(* IEC 61131-3 sources: STruCpp/tests/st-validation/function_blocks, 40 files *)

(* ---- basic_fb.st ---- *)
FUNCTION_BLOCK Counter
  VAR_INPUT increment : INT; END_VAR
  VAR_OUTPUT count : INT; END_VAR
  count := count + increment;
END_FUNCTION_BLOCK

FUNCTION_BLOCK Toggle
  VAR_OUTPUT state : BOOL; END_VAR
  state := NOT state;
END_FUNCTION_BLOCK

(* ---- fb_abstract.st ---- *)
FUNCTION_BLOCK ABSTRACT Shape
  VAR_OUTPUT area : REAL; END_VAR

  METHOD PUBLIC ABSTRACT GetArea : REAL
  END_METHOD
END_FUNCTION_BLOCK

FUNCTION_BLOCK Circle EXTENDS Shape
  VAR_INPUT radius : REAL; END_VAR

  METHOD PUBLIC GetArea : REAL
    GetArea := 3.14159 * radius * radius;
  END_METHOD

  area := THIS.GetArea();
END_FUNCTION_BLOCK

(* ---- fb_accumulator.st ---- *)
FUNCTION_BLOCK AccumulatorFB
  VAR_INPUT inc : INT; END_VAR
  VAR total : INT; END_VAR
  VAR_OUTPUT result : INT; END_VAR
  total := total + inc;
  result := total;
END_FUNCTION_BLOCK

(* ---- fb_composition.st ---- *)
FUNCTION_BLOCK Sensor
  VAR_OUTPUT value : INT; END_VAR
  value := 42;
END_FUNCTION_BLOCK

FUNCTION_BLOCK Controller
  VAR
    sensor : Sensor;
    reading : INT;
    processed : BOOL;
  END_VAR
  sensor();
  reading := sensor.value;
  processed := TRUE;
END_FUNCTION_BLOCK

(* ---- fb_constructor_defaults.st ---- *)
FUNCTION_BLOCK ConfigFB
  VAR_INPUT
    maxCount : INT;
  END_VAR
  VAR_OUTPUT
    ready : BOOL;
  END_VAR
  VAR
    counter : INT;
  END_VAR
  IF counter < maxCount THEN
    counter := counter + 1;
  END_IF;
  ready := counter >= maxCount;
END_FUNCTION_BLOCK

(* ---- fb_deep_method.st ---- *)
FUNCTION_BLOCK Inner
  VAR_INPUT seed : INT; END_VAR
  VAR_OUTPUT val : INT; END_VAR
  METHOD PUBLIC GetVal : INT
    GetVal := val + seed;
  END_METHOD
END_FUNCTION_BLOCK

FUNCTION_BLOCK Outer
  VAR
    m : Inner;
    cached : INT;
  END_VAR
  METHOD PUBLIC ReadInner : INT
    ReadInner := m.GetVal();
  END_METHOD
END_FUNCTION_BLOCK

(* ---- fb_edge_temp.st ---- *)
(* Edge inputs BOOL R_EDGE / F_EDGE (IEC 61131-3 6.6.3.2 item 13, Table 44) and
   VAR_TEMP created at each call (6.5.2.1). *)
FUNCTION_BLOCK EdgeFB
  VAR_INPUT
    Start : BOOL R_EDGE;
    Stop : BOOL F_EDGE;
    Plain : BOOL;
  END_VAR
  VAR_OUTPUT
    starts : INT;
    stops : INT;
    sawStart : BOOL;
  END_VAR
  VAR_TEMP
    t : INT;
    t2 : INT := 7;
  END_VAR
  sawStart := Start;
  IF Start THEN starts := starts + 1; END_IF;
  IF Stop THEN stops := stops + 1; END_IF;
  t := t + 1;          (* always 1: a temporary starts at its default each call *)
  t2 := t2 + t;        (* always 8 *)
  IF t <> 1 OR t2 <> 8 THEN starts := -100; END_IF;
END_FUNCTION_BLOCK

(* ---- fb_final.st ---- *)
FUNCTION_BLOCK FINAL SealedFB
  VAR_INPUT x : INT; END_VAR
  VAR_OUTPUT y : INT; END_VAR
  y := x + 1;
END_FUNCTION_BLOCK

(* ---- fb_inherit_inout.st ---- *)
(* A derived block uses its base's VAR_IN_OUT as its own (IEC 61131-3
   6.6.5.5.2 rule 2): through the in-out, in its body and around SUPER(). *)
TYPE
  IO_SET : STRUCT x : INT; END_STRUCT;
  IO_STS : STRUCT y : BOOL; n : INT; END_STRUCT;
  IO_DATA : STRUCT set : IO_SET; sts : IO_STS; simulate : BOOL; END_STRUCT;
  IO_EXTRA : STRUCT z : INT; END_STRUCT;
END_TYPE

FUNCTION_BLOCK IoBase
  VAR_IN_OUT Data : IO_DATA; END_VAR
  VAR_OUTPUT q : INT; END_VAR
  Data.sts.y := Data.set.x > 0;
  Data.sts.n := Data.sts.n + 1;
  q := Data.set.x;
END_FUNCTION_BLOCK

FUNCTION_BLOCK IoDerived EXTENDS IoBase
  VAR_IN_OUT Extra : IO_EXTRA; END_VAR
  Data.set.x := Extra.z;
  SUPER();
  IF Data.sts.y AND NOT Data.simulate THEN
    Extra.z := Extra.z + 10;
  END_IF;
END_FUNCTION_BLOCK

(* ---- fb_inheritance.st ---- *)
FUNCTION_BLOCK Base
  VAR
    _val : INT;
  END_VAR

  METHOD PUBLIC SetValue
    VAR_INPUT v : INT; END_VAR
    _val := v;
  END_METHOD

  METHOD PUBLIC GetValue : INT
    GetValue := _val;
  END_METHOD
END_FUNCTION_BLOCK

FUNCTION_BLOCK Derived EXTENDS Base
  METHOD PUBLIC DoubleIt
    _val := _val * 2;
  END_METHOD
END_FUNCTION_BLOCK

FUNCTION_BLOCK TagBase
  METHOD PUBLIC GetTag : INT
    GetTag := 1;
  END_METHOD
END_FUNCTION_BLOCK

FUNCTION_BLOCK TagDerived EXTENDS TagBase
  METHOD PUBLIC OVERRIDE GetTag : INT
    GetTag := 42;
  END_METHOD
END_FUNCTION_BLOCK

(* ---- fb_interface_vars.st ---- *)
INTERFACE I_MOTOR_BASE
  METHOD Id : INT
  END_METHOD
END_INTERFACE

INTERFACE I_MOTOR EXTENDS I_MOTOR_BASE
  METHOD IsRunning : BOOL
  END_METHOD
  METHOD Start
    VAR_INPUT Speed : REAL; END_VAR
  END_METHOD
END_INTERFACE

INTERFACE I_SPEED EXTENDS I_MOTOR_BASE
  METHOD Speed : REAL
  END_METHOD
END_INTERFACE

FUNCTION_BLOCK MotorDol IMPLEMENTS I_MOTOR
  VAR running : BOOL; END_VAR
  METHOD PUBLIC Id : INT
    Id := 1;
  END_METHOD
  METHOD PUBLIC IsRunning : BOOL
    IsRunning := running;
  END_METHOD
  METHOD PUBLIC Start
    VAR_INPUT Speed : REAL; END_VAR
    running := TRUE;
  END_METHOD
END_FUNCTION_BLOCK

FUNCTION_BLOCK MotorVsd IMPLEMENTS I_MOTOR, I_SPEED
  VAR spd : REAL; END_VAR
  METHOD PUBLIC Id : INT
    Id := 2;
  END_METHOD
  METHOD PUBLIC IsRunning : BOOL
    IsRunning := spd > 0.0;
  END_METHOD
  METHOD PUBLIC Start
    VAR_INPUT Speed : REAL; END_VAR
    spd := Speed;
  END_METHOD
  METHOD PUBLIC Speed : REAL
    Speed := spd;
  END_METHOD
END_FUNCTION_BLOCK

FUNCTION_BLOCK MotorVsdFast EXTENDS MotorVsd
  METHOD PUBLIC OVERRIDE Id : INT
    Id := 3;
  END_METHOD
END_FUNCTION_BLOCK

FUNCTION_BLOCK Pump
  VAR_INPUT Demand : BOOL; Motor : I_MOTOR; END_VAR
  VAR_OUTPUT Run : BOOL; Valid : BOOL; END_VAR
  Valid := Motor <> NULL;
  IF NOT Valid THEN
    Run := FALSE;
    RETURN;
  END_IF;
  IF Demand THEN Motor.Start(Speed := 50.0); END_IF;
  Run := Motor.IsRunning();
END_FUNCTION_BLOCK

FUNCTION_BLOCK Station
  VAR_IN_OUT Motors : ARRAY[*] OF I_MOTOR; END_VAR
  VAR_OUTPUT Running : INT; IdSum : INT; END_VAR
  VAR i : DINT; END_VAR
  Running := 0;
  IdSum := 0;
  FOR i := LOWER_BOUND(Motors, 1) TO UPPER_BOUND(Motors, 1) DO
    IF Motors[i] <> NULL THEN
      IdSum := IdSum + Motors[i].Id();
      IF Motors[i].IsRunning() THEN Running := Running + 1; END_IF;
    END_IF;
  END_FOR;
END_FUNCTION_BLOCK

FUNCTION MotorId : INT
  VAR_INPUT m : I_MOTOR_BASE; END_VAR
  IF m = NULL THEN
    MotorId := -1;
  ELSE
    MotorId := m.Id();
  END_IF;
END_FUNCTION

(* ---- fb_interfaces.st ---- *)
INTERFACE IMovable
  METHOD MoveTo : BOOL
    VAR_INPUT x : INT; y : INT; END_VAR
  END_METHOD
END_INTERFACE

FUNCTION_BLOCK Robot IMPLEMENTS IMovable
  VAR
    posX : INT;
    posY : INT;
  END_VAR

  METHOD PUBLIC MoveTo : BOOL
    VAR_INPUT x : INT; y : INT; END_VAR
    posX := x;
    posY := y;
    MoveTo := TRUE;
  END_METHOD
END_FUNCTION_BLOCK

(* ---- fb_method_collision.st ---- *)
FUNCTION_BLOCK Adder
  VAR_INPUT x : INT; END_VAR
  METHOD PUBLIC Compute : INT
    Compute := x + 100;
  END_METHOD
END_FUNCTION_BLOCK

FUNCTION_BLOCK Doubler
  VAR_INPUT x : INT; END_VAR
  METHOD PUBLIC Compute : INT
    Compute := x * 2;
  END_METHOD
END_FUNCTION_BLOCK

(* ---- fb_method_names.st ---- *)
(* Methods of a block: its own, an inherited one, and prototypes of an interface
   it implements through EXTENDS. A variable cannot share a method's name
   (IEC 61131-3 6.6.5.5.5 rule 2), so the outputs carry their own names. *)
INTERFACE I_A
  METHOD Good : BOOL END_METHOD
END_INTERFACE
INTERFACE I_B EXTENDS I_A
  METHOD Total : LREAL END_METHOD
END_INTERFACE
FUNCTION_BLOCK F IMPLEMENTS I_B
  VAR_OUTPUT IsGood : BOOL; TotalOut : LREAL; OwnOut : INT; END_VAR
  METHOD PUBLIC Good : BOOL Good := TRUE; END_METHOD
  METHOD PUBLIC Total : LREAL Total := 1.0; END_METHOD
  METHOD PUBLIC Own : INT Own := 7; END_METHOD
  IsGood := THIS.Good(); TotalOut := THIS.Total(); OwnOut := THIS.Own();
END_FUNCTION_BLOCK
FUNCTION_BLOCK G EXTENDS F
  VAR_OUTPUT Sum : LREAL; END_VAR
  SUPER();
  Sum := TotalOut + THIS.Total();
END_FUNCTION_BLOCK

(* ---- fb_methods.st ---- *)
FUNCTION_BLOCK Motor
  VAR
    _speed : INT;
    _running : BOOL;
  END_VAR

  METHOD PUBLIC Start
    _running := TRUE;
  END_METHOD

  METHOD PUBLIC Stop
    _running := FALSE;
    _speed := 0;
  END_METHOD

  METHOD PUBLIC SetSpeed
    VAR_INPUT newSpeed : INT; END_VAR
    IF _running THEN
      _speed := newSpeed;
    END_IF;
  END_METHOD

  METHOD PUBLIC GetSpeed : INT
    GetSpeed := _speed;
  END_METHOD

  METHOD PUBLIC IsRunning : BOOL
    IsRunning := _running;
  END_METHOD
END_FUNCTION_BLOCK

(* ---- fb_output_capture.st ---- *)
FUNCTION_BLOCK Calculator
  VAR_INPUT a : INT; b : INT; END_VAR
  VAR_OUTPUT sum : INT; product : INT; END_VAR
  sum := a + b;
  product := a * b;
END_FUNCTION_BLOCK

(* ---- fb_properties.st ---- *)
FUNCTION_BLOCK MotorProp
  VAR _speed : INT; END_VAR

  PROPERTY Speed : INT
    GET
      Speed := _speed;
    END_GET
    SET
      IF Speed > 100 THEN
        _speed := 100;
      ELSE
        _speed := Speed;
      END_IF;
    END_SET
  END_PROPERTY
END_FUNCTION_BLOCK

FUNCTION_BLOCK ControllerProp
  VAR motor : MotorProp; END_VAR
END_FUNCTION_BLOCK

(* ---- fb_state.st ---- *)
FUNCTION_BLOCK Accumulator
  VAR_INPUT value : INT; END_VAR
  VAR_OUTPUT total : INT; END_VAR
  VAR callCount : INT; END_VAR
  total := total + value;
  callCount := callCount + 1;
END_FUNCTION_BLOCK

FUNCTION_BLOCK MaxTracker
  VAR_INPUT input : INT; END_VAR
  VAR_OUTPUT maxValue : INT; END_VAR
  IF input > maxValue THEN
    maxValue := input;
  END_IF;
END_FUNCTION_BLOCK

(* ---- fb_super_iec.st ---- *)
(* Function block inheritance in the IEC forms (IEC 61131-3 6.6.7.2.7-11):
   SUPER() runs the base body, calls bind dynamically, SUPER.m(), THIS. *)
INTERFACE I_KIND
  METHOD Kind : INT
  END_METHOD
END_INTERFACE

FUNCTION_BLOCK ABSTRACT BaseFB IMPLEMENTS I_KIND
  VAR_INPUT a : INT; END_VAR
  VAR_OUTPUT x : INT; END_VAR
  VAR PROTECTED calls : INT; END_VAR
  VAR PRIVATE secret : INT; END_VAR
  METHOD PUBLIC Kind : INT
    Kind := 1;
  END_METHOD
  METHOD PUBLIC ABSTRACT Scale : INT
  END_METHOD
  METHOD PROTECTED Bump
    calls := calls + 1;
  END_METHOD
  x := a + 1;
  THIS.Bump();
END_FUNCTION_BLOCK

FUNCTION_BLOCK Derived1 EXTENDS BaseFB
  VAR_INPUT b : INT; END_VAR
  METHOD PUBLIC OVERRIDE Kind : INT
    Kind := SUPER.Kind() + 10;
  END_METHOD
  METHOD PUBLIC Scale : INT
    Scale := 3;
  END_METHOD
  SUPER();
  x := THIS.Scale() * x + b;
END_FUNCTION_BLOCK

FUNCTION_BLOCK FINAL Derived2 EXTENDS Derived1
  VAR_IN_OUT c : INT; END_VAR
  METHOD PUBLIC FINAL OVERRIDE Kind : INT
    Kind := 20;
  END_METHOD
  SUPER();
  c := x;
END_FUNCTION_BLOCK

FUNCTION_BLOCK Runner
  VAR_IN_OUT inst : Derived1; END_VAR
  inst(a := 1, b := 2);
END_FUNCTION_BLOCK

FUNCTION KindOf : INT
  VAR_INPUT k : I_KIND; END_VAR
  IF k <> NULL THEN KindOf := k.Kind(); ELSE KindOf := -1; END_IF;
END_FUNCTION

FUNCTION_BLOCK Derived3 EXTENDS Derived1
  SUPER();
  x := x + 1000;
END_FUNCTION_BLOCK
INTERFACE I_ROOM
  METHOD DAYTIME END_METHOD
  METHOD NIGHTTIME END_METHOD
END_INTERFACE
FUNCTION_BLOCK ROOM_CTRL
  VAR_INPUT RM : I_ROOM; Night : BOOL; END_VAR
  IF RM = NULL THEN RETURN; END_IF;
  IF Night THEN RM.NIGHTTIME(); ELSE RM.DAYTIME(); END_IF;
END_FUNCTION_BLOCK
FUNCTION_BLOCK LIGHTROOM IMPLEMENTS I_ROOM
  VAR PUBLIC LIGHT : BOOL; END_VAR
  VAR PROTECTED level : INT; END_VAR
  METHOD PUBLIC DAYTIME LIGHT := FALSE; END_METHOD
  METHOD PUBLIC NIGHTTIME LIGHT := TRUE; level := 1; END_METHOD
  METHOD PROTECTED Dim level := level - 1; END_METHOD
END_FUNCTION_BLOCK
FUNCTION_BLOCK LIGHT2ROOM EXTENDS LIGHTROOM IMPLEMENTS I_ROOM
  VAR PUBLIC LIGHT2 : BOOL; END_VAR
  VAR ctrl : ROOM_CTRL; END_VAR
  VAR_INPUT Night : BOOL; END_VAR
  METHOD PUBLIC OVERRIDE DAYTIME
    SUPER.DAYTIME();
    LIGHT2 := TRUE;
  END_METHOD
  METHOD PUBLIC OVERRIDE NIGHTTIME
    SUPER.NIGHTTIME();
    LIGHT2 := FALSE;
    level := level + 10;
    THIS.Dim();
  END_METHOD
  ctrl(RM := THIS, Night := Night);
END_FUNCTION_BLOCK
FUNCTION_BLOCK ABSTRACT SHAPE
  VAR_OUTPUT area : REAL; END_VAR
  METHOD PUBLIC ABSTRACT Calc : REAL END_METHOD
  area := THIS.Calc();
END_FUNCTION_BLOCK
FUNCTION_BLOCK SQUARE EXTENDS SHAPE
  VAR_INPUT side : REAL; END_VAR
  METHOD PUBLIC Calc : REAL Calc := side * side; END_METHOD
  SUPER();
END_FUNCTION_BLOCK

(* ---- fb_this_super.st ---- *)
FUNCTION_BLOCK ComputeBase
  VAR_INPUT value : INT; END_VAR
  VAR_OUTPUT result : INT; END_VAR

  METHOD PUBLIC Compute : INT
    Compute := value * 2;
  END_METHOD

  result := THIS.Compute();
END_FUNCTION_BLOCK

(* ---- test_basic_fb.st ---- *)
TEST 'Counter increments by specified amount'
  VAR c : Counter; END_VAR
  c(increment := 5);
  ASSERT_EQ(c.count, 5);
  c(increment := 3);
  ASSERT_EQ(c.count, 8);
END_TEST

TEST 'Counter starts at zero'
  VAR c : Counter; END_VAR
  ASSERT_EQ(c.count, 0);
END_TEST

TEST 'Two counters are independent'
  VAR a : Counter; b : Counter; END_VAR
  a(increment := 10);
  b(increment := 20);
  ASSERT_EQ(a.count, 10);
  ASSERT_EQ(b.count, 20);
END_TEST

TEST 'Toggle alternates state'
  VAR t : Toggle; END_VAR
  ASSERT_FALSE(t.state);
  t();
  ASSERT_TRUE(t.state);
  t();
  ASSERT_FALSE(t.state);
  t();
  ASSERT_TRUE(t.state);
END_TEST

(* ---- test_fb_abstract.st ---- *)
TEST 'Concrete class computes area'
  VAR c : Circle; END_VAR
  c(radius := 2.0);
  ASSERT_NEAR(c.area, 12.566, 0.01);
END_TEST

(* ---- test_fb_accumulator.st ---- *)
TEST 'Accumulator preserves state across calls'
  VAR acc : AccumulatorFB; END_VAR
  acc(inc := 3);
  ASSERT_EQ(acc.result, 3);
  acc(inc := 3);
  ASSERT_EQ(acc.result, 6);
  acc(inc := 3);
  ASSERT_EQ(acc.result, 9);
END_TEST

(* ---- test_fb_composition.st ---- *)
TEST 'FB composition: Controller reads Sensor'
  VAR ctrl : Controller; END_VAR
  ctrl();
  ASSERT_EQ(ctrl.reading, 42);
  ASSERT_TRUE(ctrl.processed);
END_TEST

TEST 'FB composition: nested FB invoked'
  VAR ctrl : Controller; END_VAR
  ctrl();
  ASSERT_EQ(ctrl.sensor.value, 42);
END_TEST

(* ---- test_fb_constructor_defaults.st ---- *)
TEST 'FB input not ready after single call with high limit'
  VAR cfg : ConfigFB; END_VAR
  cfg(maxCount := 100);
  ASSERT_FALSE(cfg.ready);
END_TEST

TEST 'FB input ready when limit is 1'
  VAR cfg : ConfigFB; END_VAR
  cfg(maxCount := 1);
  ASSERT_TRUE(cfg.ready);
END_TEST

(* ---- test_fb_deep_method.st ---- *)
TEST 'Method in Outer calls Inner.GetVal()'
  VAR ctrl : Outer; result : INT; END_VAR
  ctrl.m.seed := 10;
  ctrl.m.val := 5;
  result := ctrl.ReadInner();
  ASSERT_EQ(result, 15);
END_TEST

(* ---- test_fb_edge_temp.st ---- *)
TEST 'rising edge once per transition, held TRUE at first call is an edge'
  VAR e : EdgeFB; END_VAR
  e(Start := TRUE, Stop := TRUE);
  ASSERT_EQ(e.starts, 1);
  e(Start := TRUE);
  ASSERT_EQ(e.starts, 1);
  ASSERT_FALSE(e.sawStart);
  e();
  e();
  ASSERT_EQ(e.starts, 1);
  e(Start := FALSE);
  e(Start := TRUE);
  ASSERT_EQ(e.starts, 2);
  ASSERT_TRUE(e.sawStart);
  ASSERT_TRUE(e.Start);
END_TEST
TEST 'falling edge, input FALSE at first call is an edge (Table 44 note)'
  VAR e : EdgeFB; END_VAR
  e(Stop := FALSE);
  ASSERT_EQ(e.stops, 1);
  e(Stop := FALSE);
  ASSERT_EQ(e.stops, 1);
  e(Stop := TRUE);
  ASSERT_EQ(e.stops, 1);
  e(Stop := FALSE);
  ASSERT_EQ(e.stops, 2);
END_TEST

(* ---- test_fb_final.st ---- *)
TEST 'FINAL FB computes correctly'
  VAR s : SealedFB; END_VAR
  s(x := 42);
  ASSERT_EQ(s.y, 43);
END_TEST

(* ---- test_fb_inherit_inout.st ---- *)
TEST 'derived body reads and writes the base in-out, both in-outs bound'
  VAR d : IoDerived; data : IO_DATA; extra : IO_EXTRA; END_VAR
  extra.z := 3;
  d(Data := data, Extra := extra);
  ASSERT_EQ(data.set.x, 3);
  ASSERT_TRUE(data.sts.y);
  ASSERT_EQ(data.sts.n, 1);
  ASSERT_EQ(d.q, 3);
  ASSERT_EQ(extra.z, 13);
  data.simulate := TRUE;
  d(Data := data, Extra := extra);
  ASSERT_EQ(data.set.x, 13);
  ASSERT_EQ(data.sts.n, 2);
  ASSERT_EQ(extra.z, 13);
END_TEST

(* ---- test_fb_inheritance.st ---- *)
TEST 'Derived inherits base methods'
  VAR d : Derived; END_VAR
  d.SetValue(v := 10);
  ASSERT_EQ(d.GetValue(), 10);
END_TEST

TEST 'Derived can add new methods'
  VAR d : Derived; END_VAR
  d.SetValue(v := 5);
  d.DoubleIt();
  ASSERT_EQ(d.GetValue(), 10);
END_TEST

TEST 'Override dispatch returns derived value'
  VAR d : TagDerived; result : INT; END_VAR
  result := d.GetTag();
  ASSERT_EQ(result, 42);
END_TEST

(* ---- test_fb_interface_vars.st ---- *)
TEST 'pump runs either motor type through its interface input'
  VAR dol : MotorDol; vsd : MotorVsd; p1 : Pump; p2 : Pump; END_VAR
  p1(Demand := TRUE, Motor := dol);
  p2(Demand := TRUE, Motor := vsd);
  ASSERT_TRUE(p1.Valid);
  ASSERT_TRUE(p1.Run);
  ASSERT_TRUE(p2.Run);
  ASSERT_EQ(vsd.Speed(), 50.0);
END_TEST

TEST 'unassigned interface input is NULL'
  VAR p : Pump; END_VAR
  p(Demand := TRUE);
  ASSERT_FALSE(p.Valid);
  ASSERT_FALSE(p.Run);
END_TEST

TEST 'interface variables compare by instance'
  VAR dol : MotorDol; other : MotorDol; a : I_MOTOR; b : I_MOTOR := dol; END_VAR
  ASSERT_TRUE(a = NULL);
  a := dol;
  ASSERT_TRUE(a = b);
  a := other;
  ASSERT_TRUE(a <> b);
END_TEST

TEST 'derived interface to base, overriding method through it'
  VAR fast : MotorVsdFast; m : I_MOTOR; base : I_MOTOR_BASE; END_VAR
  m := fast;
  base := m;
  ASSERT_EQ(MotorId(m := base), 3);
  ASSERT_EQ(MotorId(m := NULL), -1);
END_TEST

TEST 'array of interface references as an in-out'
  VAR dol : MotorDol; vsd : MotorVsd; st : Station; ms : ARRAY[1..3] OF I_MOTOR; END_VAR
  dol.Start(Speed := 1.0);
  ms[1] := dol;
  ms[3] := vsd;
  st(Motors := ms);
  ASSERT_EQ(st.Running, 1);
  ASSERT_EQ(st.IdSum, 3);
  ASSERT_TRUE(ms[1].IsRunning());
END_TEST

TEST 'assignment attempt'
  VAR dol : MotorDol; vsd : MotorVsd; b : I_MOTOR_BASE; s : I_SPEED; END_VAR
  b := dol;
  s ?= b;
  ASSERT_TRUE(s = NULL);
  b := vsd;
  s ?= b;
  ASSERT_TRUE(s <> NULL);
  s ?= NULL;
  ASSERT_TRUE(s = NULL);
  s ?= vsd;
  ASSERT_EQ(s.Id(), 2);
END_TEST

(* ---- test_fb_interfaces.st ---- *)
TEST 'FB implements interface method'
  VAR bot : Robot; ok : BOOL; END_VAR
  ok := bot.MoveTo(x := 10, y := 20);
  ASSERT_TRUE(ok);
  ASSERT_EQ(bot.posX, 10);
  ASSERT_EQ(bot.posY, 20);
END_TEST

(* ---- test_fb_method_collision.st ---- *)
TEST 'Two FBs with same method name dispatch correctly'
  VAR a : Adder; d : Doubler; r1, r2 : INT; END_VAR
  a.x := 5;
  d.x := 5;
  r1 := a.Compute();
  r2 := d.Compute();
  ASSERT_EQ(r1, 105);
  ASSERT_EQ(r2, 10);
END_TEST

(* ---- test_fb_method_names.st ---- *)
TEST 'methods of a block, inherited and through interfaces'
  VAR f : F; g : G; m : I_A; END_VAR
  f();
  ASSERT_TRUE(f.IsGood);
  ASSERT_EQ(f.TotalOut, 1.0);
  ASSERT_EQ(f.OwnOut, 7);
  g();
  ASSERT_EQ(g.Sum, 2.0);
  m := g;
  ASSERT_TRUE(m.Good());
END_TEST

(* ---- test_fb_methods.st ---- *)
TEST 'Motor starts and stops'
  VAR m : Motor; END_VAR
  ASSERT_FALSE(m.IsRunning());
  m.Start();
  ASSERT_TRUE(m.IsRunning());
  m.Stop();
  ASSERT_FALSE(m.IsRunning());
END_TEST

TEST 'Motor speed only changes when running'
  VAR m : Motor; END_VAR
  m.SetSpeed(newSpeed := 100);
  ASSERT_EQ(m.GetSpeed(), 0);
  m.Start();
  m.SetSpeed(newSpeed := 750);
  ASSERT_EQ(m.GetSpeed(), 750);
END_TEST

TEST 'Motor stop resets speed'
  VAR m : Motor; END_VAR
  m.Start();
  m.SetSpeed(newSpeed := 500);
  m.Stop();
  ASSERT_EQ(m.GetSpeed(), 0);
END_TEST

(* ---- test_fb_output_capture.st ---- *)
TEST 'FB output capture with => syntax'
  VAR calc : Calculator; mySum, myProduct : INT; END_VAR
  calc(a := 5, b := 3, sum => mySum, product => myProduct);
  ASSERT_EQ(mySum, 8);
  ASSERT_EQ(myProduct, 15);
END_TEST

(* ---- test_fb_properties.st ---- *)
TEST 'Property setter and getter work'
  VAR m : MotorProp; x : INT; END_VAR
  m.Speed := 75;
  x := m.Speed;
  ASSERT_EQ(x, 75);
END_TEST

TEST 'Property setter clamps above threshold'
  VAR m : MotorProp; x : INT; END_VAR
  m.Speed := 200;
  x := m.Speed;
  ASSERT_EQ(x, 100);
END_TEST

(* ---- test_fb_state.st ---- *)
TEST 'Accumulator accumulates over multiple calls'
  VAR acc : Accumulator; END_VAR
  acc(value := 10);
  acc(value := 20);
  acc(value := 30);
  ASSERT_EQ(acc.total, 60);
END_TEST

TEST 'Accumulator internal state tracks calls'
  VAR acc : Accumulator; END_VAR
  acc(value := 1);
  acc(value := 1);
  ASSERT_EQ(acc.callCount, 2);
END_TEST

TEST 'MaxTracker tracks maximum input'
  VAR mt : MaxTracker; END_VAR
  mt(input := 5);
  ASSERT_EQ(mt.maxValue, 5);
  mt(input := 3);
  ASSERT_EQ(mt.maxValue, 5);
  mt(input := 8);
  ASSERT_EQ(mt.maxValue, 8);
  mt(input := 1);
  ASSERT_EQ(mt.maxValue, 8);
END_TEST

(* ---- test_fb_super_iec.st ---- *)
TEST 'super body once'
  VAR d : Derived1; END_VAR
  d(a := 123, b := 1);
  ASSERT_EQ(d.x, 373);

END_TEST
TEST 'chain'
  VAR d : Derived2; v : INT; END_VAR
  d(a := 1, b := 2, c := v);
  ASSERT_EQ(d.x, 8);
  ASSERT_EQ(v, 8);
END_TEST
TEST 'override and interface'
  VAR d1 : Derived1; d2 : Derived2; END_VAR
  ASSERT_EQ(KindOf(k := d1), 11);
  ASSERT_EQ(KindOf(k := d2), 20);
END_TEST
TEST 'dynamic body binding through in-out of base type'
  VAR d3 : Derived3; r : Runner; END_VAR
  r(inst := d3);
  ASSERT_EQ(d3.x, 1008);
END_TEST

TEST 'IEC example: LIGHT2ROOM with SUPER, THIS passed to an interface input'
  VAR r : LIGHT2ROOM; c : ROOM_CTRL; END_VAR
  c(RM := r, Night := TRUE);
  ASSERT_TRUE(r.LIGHT);
  ASSERT_FALSE(r.LIGHT2);
  c(RM := r, Night := FALSE);
  ASSERT_FALSE(r.LIGHT);
  ASSERT_TRUE(r.LIGHT2);
  r(Night := TRUE);
  ASSERT_TRUE(r.LIGHT);
  ASSERT_FALSE(r.LIGHT2);
END_TEST
TEST 'abstract method implemented in derived, base body via SUPER'
  VAR s : SQUARE; END_VAR
  s(side := 3.0);
  ASSERT_EQ(s.area, 9.0);
END_TEST

(* ---- test_fb_this_super.st ---- *)
TEST 'Base uses THIS to call own method'
  VAR b : ComputeBase; END_VAR
  b(value := 5);
  ASSERT_EQ(b.result, 10);
END_TEST
